// TIA Portal project "Project2_Sim_Correction" (V17)

(* hardware
DEVICE "PC_STATION"  SIMATIC PC station
   slot 0: "PC station"  Rail  SIMATIC PC-Station  V1.0
      slot 125: "Stationmanager"  Station_Manager  V6.0.4
   slot 1: "IE general_1"  IE General  IE_CP  V8.2.0
      slot 1: "PROFINET interface"  IEGeneral.Interface.8.2.0
   slot 3: "HMI_RT_1"  WinCC RT Advanced  6AV2 104-0xxxx-xxxx  17.0.0.0
      slot 33792: "Computer interface"  Host interface
DEVICE "S7-1500/ET200MP station_1"  S7-1500 station
   slot 0: "Rail_0"  Rack  6ES7 590-1***0-0AA0
   slot 1: "PLC_1"  CPU 1511-1 PN  6ES7 511-1AK02-0AB0  V2.9
      slot 3: "CPU display_1"  6ES7591-1AA00-0AA0
      slot 32768: "PROFINET interface_1"  X1
         slot 32769: "Port_1"  X1 P1
         slot 32770: "Port_2"  X1 P2
      slot 34817: "Virtual CP interface port_1"  Virtual CP interface port  Virtual CP interface port
*)

// ===== PLC "PLC_1"  CPU 1511-1 PN =====

VAR_GLOBAL   // PLC tag table "New Table"
   "Level_Sensor" AT %MD2 : Real;
   "Manual_Mode" AT %M0.1 : Bool;
   "Start_Button" AT %M0.2 : Bool;
   "Stop_Button" AT %M0.3 : Bool;
   "Inlet_Valve" AT %M1.0 : Bool;
   "Outlet_Pump" AT %M1.1 : Bool;
   "High_Level" AT %MD0 : Real;
   "Low_Level" AT %MD1 : Real;
   "Alarm" AT %M1.2 : Bool;
END_VAR

ORGANIZATION_BLOCK "Main"   // OB1, LAD, ProgramCycle
TITLE = "Main Program Sweep (Cycle)"
{ S7_Optimized_Access := 'TRUE' }
VERSION : 0.1
   VAR_INPUT
      Initial_Call : Bool;   // Initial call of this OB
      Remanence : Bool;   // =True, if remanent data are available
   END_VAR
BEGIN

REGION Network 1
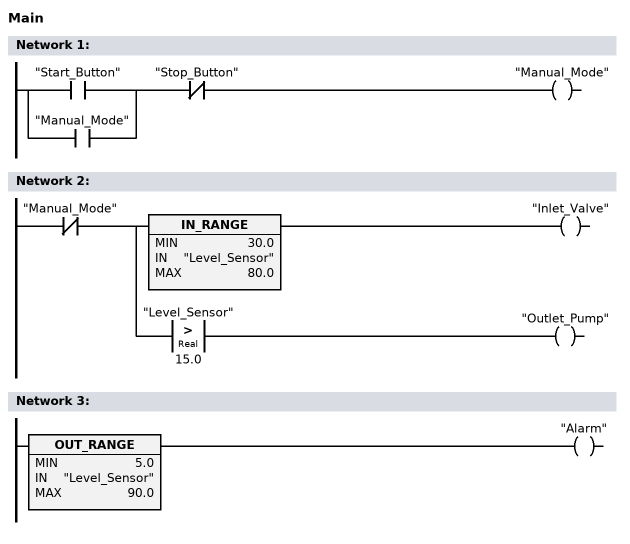
   RUNG wire#powerrail
      Contact( "Start_Button" )
      wire#w1
      I_Contact( "Stop_Button" )
      Coil( "Manual_Mode" )
   END_RUNG
   RUNG wire#powerrail
      Contact( "Manual_Mode" )
   END_RUNG wire#w1
   // the same network as SCL:
   "Manual_Mode" := ("Start_Button" OR "Manual_Mode") AND NOT "Stop_Button";
END_REGION

REGION Network 2
   RUNG wire#powerrail
      I_Contact( "Manual_Mode" )
      wire#w1
      { S7_Templates := "SrcType := Real" } InRange(min := 30.0, in := "Level_Sensor", max := 80.0)
      Coil( "Inlet_Valve" )
   END_RUNG
   RUNG wire#w1
      { S7_Templates := "SrcType := Real" } GT_Contact(in1 := "Level_Sensor", in2 := 15.0)
      Coil( "Outlet_Pump" )
   END_RUNG
   // the same network as SCL:
   "Inlet_Valve" := NOT "Manual_Mode" AND (30.0 <= "Level_Sensor") AND ("Level_Sensor" <= 80.0);
   "Outlet_Pump" := NOT "Manual_Mode" AND ("Level_Sensor" > 15.0);
END_REGION

REGION Network 3
   "Alarm" := ("Level_Sensor" < 5.0) OR ("Level_Sensor" > 90.0);
END_REGION
END_ORGANIZATION_BLOCK

(* ===== HMI "HMI_RT_1" =====
system functions are stored by id; their names below are inferred from use
connection "HMI_Connection_1": ETHERNET, S7_1500_OMS

HMI tags "Tag table_1"
   "HMI_Start" : Bool = PLC Start_Button AT %M0.2, 100 ms
      on ChangeValue: SetBit("HMI_Start")
   "HMI_Stop" : Bool = PLC Stop_Button AT %M0.3, 100 ms
   "HMI_level_sensor" : Real = PLC Level_Sensor AT %MD2, 100 ms
   "HMI_inlet_valve" : Bool = PLC Inlet_Valve AT %M1.0, 100 ms
   "HMI_outlet_pump" : Bool = PLC Outlet_Pump AT %M1.1, 100 ms

screen "Screen_1" 800x480
   Switch "Switch_1" at 34,39 size 120x88; CaptionText 'Start'; TextOff 'OFF'; TextOn 'ON'
      ProcessValue <- "HMI_Start"
      on SwitchOn: SetBit("HMI_Start")
      on SwitchOff: ResetBit("HMI_Start")
   Switch "Switch_2" at 34,202 size 120x88; TextOn 'ON'; CaptionText 'Stop'; TextOff 'OFF'
      ProcessValue <- "HMI_Stop"
      on SwitchOn: SetBit("HMI_Stop")
      on SwitchOff: ResetBit("HMI_Stop")
   Gauge "Gauge_1" at 290,90 size 200x200; CaptionText 'SIMATIC'; UnitText 'Unit'
      ProcessValue <- "HMI_level_sensor"
   GraphicView "Graphic view_1" at 588,111 size 113x140; Picture "Graphic_3"
      Appearance <- "HMI_outlet_pump"
   GraphicView "Graphic view_2" at 793,113 size 153x138; Picture "Graphic_4"
      Appearance <- "HMI_inlet_valve"
   TextField "Text field_2" at 815,64 size 104x47; Text 'Valve'
   TextField "Text field_1" at 588,60 size 109x47; Text 'Pump'
   TextField "Text field_3" at 283,35 size 235x47; Text 'Level Sensor'
   Rectangle "Rectangle_1" at 49,133 size 96x48
      Appearance <- "HMI_Start"
   Rectangle "Rectangle_2" at 49,295 size 96x48
      Appearance <- "HMI_Stop"
*)